(* PLC project roundcam, Dassault Systèmes ControlBuild 2024x *)
(* stored: creationDateTime 2023-10-03T11:13:15-01:00 *)

(* This module simulates the behaviour of a round cam *)
FUNCTION_BLOCK equipment_library.roundcam
  VAR_INPUT
    rotationSpeedDegS : REAL := 0.0;
  END_VAR
  VAR_OUTPUT
    angleRotationDeg : REAL := 0.0;
    angleRotationRad : REAL := 0.0;
    angle_modulo : REAL := 0.0;
  END_VAR
  VAR
    firstCycle : BOOL := false;
    incrementRotation : REAL := 0.0;
  END_VAR
  VAR CONSTANT
    initAngle : REAL := 0.0;
    modulo : REAL := 1000.0;
  END_VAR
  VAR
    d_locking : BOOL := false;
    v_d_locking : BOOL := false;
  END_VAR


ACTION C_source_code:
/* ----------------------------------------------------------------	*/
/* Author : 3DS								*/
/* Update date : October 2017						*/
/* ----------------------------------------------------------------	*/
/* This module simulate the behaviour of a cam 	.			*/
/* The position of the cam goes from 0 to 360 with	*/
/* the given rotation speed.						*/
/*										*/
/* nota : - the starting position is forced by initAngle.		*/
/*	   - the speed setpoint can be set in				*/
/*		- degree per second	(rotationSpeedDegS)			*/
/* ----------------------------------------------------------------	*/

/* Declaration of variables which don't need to be visualized during simulation */

/* ----------------------------------------------------------------	*/
/* Initialization of the position of the cam for the first step of	*/
/* simulation.								*/
/* ----------------------------------------------------------------	*/
if (! firstCycle) {
	if (initAngle > 360 ) angleRotationDeg  = 360 ;
	else
		if (initAngle < 0) angleRotationDeg  = 0;
		else angleRotationDeg  = initAngle;

	firstCycle = 1;
}

/* ----------------------------------------------------------------	*/
/* Rotation and translation (height of cam)				*/
/* ----------------------------------------------------------------	*/
if ((!d_locking) && ((rotationSpeedDegS!=0.0)||(rotationSpeedDegS!=0.0))) {

	/* compute the increment of rotation according to the clock of simulation	*/

	incrementRotation= rotationSpeedDegS * (CLOCK_PERIOD /1000000.0);
	/* compute the angle of rotation (degrees)	*/
	angleRotationDeg = angleRotationDeg  + incrementRotation;
	if (angleRotationDeg  > 360 ) {angleRotationDeg  -= 360 ;}
	if (angleRotationDeg  < -360 ) {angleRotationDeg  += 360 ;}
}

/* Conversion deg in Radians  */		
angleRotationRad = angleRotationDeg * 0.03491;
angle_modulo = (angleRotationDeg *modulo) / 360.0;
END_ACTION
END_FUNCTION_BLOCK
